TYPE "MES_Msg_Send_Err"
VERSION : 0.1
// Block: MES_Msg_Send_Err
   STRUCT
      TimeOut_ACK : Bool;
      Buffer_Pop : Struct
         Presence : Bool;
         Code : DInt;
      END_STRUCT;
      Msg_NotAccepted : "MES_Err_&_Msg";
   END_STRUCT;

END_TYPE
